{attribute 'qualified_only'}
{attribute 'strict'}
TYPE ReceiveStatus :
(
	WAITING,
	RECEIVING,
	DONE,
	FAIL,
	TIMEOUT
) := RECEIVING;
END_TYPE

(* stored: Version 1.1.0.1, ProductVersion 3.1.4024.12
   DUT ReceiveStatus: Id {80f09e3c-232b-43ec-ad29-220620fbb644} *)
